Yaskawa INFORM job: HOME.JBI

/JOB
//NAME HOME
//POS
///NPOS 0,0,0,5,0,0
///TOOL 0
///POSTYPE PULSE
///PULSE
P00000=4209,-7192,-5593,1580,-64891,83596
P00001=55242,26922,11446,1601,-60437,64378
P00002=55242,35623,-7881,1830,-43902,63991
P00004=-47424,25138,-17957,938,-40698,102661
P00005=56012,31125,28227,2771,-69762,62996
//INST
///DATE 2024/08/21 18:20
///ATTR SC,RW
///GROUP1 RB1
NOP
IFTHENEXP I010=12
	 PULSE OT#(6)
	 MOVL P002 V=I003
	 MOVJ P001 VJ=I000
	 MOVJ P000 VJ=I000
ENDIF
IFTHENEXP I010=11
	 MOVJ P001 VJ=I000
	 MOVJ P000 VJ=I000
ENDIF
IFTHENEXP I011=12
	 PULSE OT#(6)
	 MOVL P005 V=I003
	 MOVJ P004 VJ=I000
	 MOVJ P000 VJ=I000
ENDIF
IFTHENEXP I011=11
	 MOVJ P004 VJ=I000
	 MOVJ P000 VJ=I000
ENDIF
IFTHENEXP I010<>11 ANDEXP B010<>12
	 MOVJ P000 VJ=I000
ENDIF
IFTHENEXP I011<>11 ANDEXP B011<>12
	 MOVJ P000 VJ=I000
ENDIF
CALL JOB:MATER
END
